{attribute 'qualified_only'}
{attribute 'strict'}
TYPE E_Direction :
(
	Right_Forward_Up,
	Left_Back_Down
);
END_TYPE

(* stored: Version 1.1.0.1, ProductVersion 3.1.4024.11
   DUT E_Direction: Id {eafedf04-7bde-4acc-a364-f68cb504bdaa} *)
